Fanuc KAREL source: KB00163.KL

PROGRAM KB00163
%NOLOCKGROUP
VAR
  P1: FILE
  P2: INTEGER
BEGIN
  P2 = 1
  SET_FILE_ATR(P1, P2)
END KB00163
